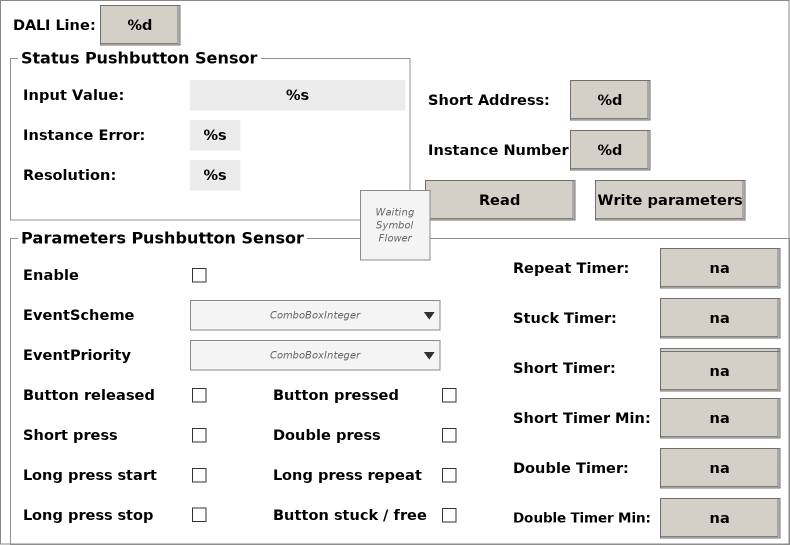
VISUALIZATION Visu_Part301PushButton  // 790x545
    GroupBox (10,230 780x315), "Parameters Pushbutton Sensor"
        Button (650,268 120x40), "%d ms", text variable: DALI_Commissioning.fbPart301PushButton.nDoubleMin
        Button (650,268 120x40), "na", invisible if: Not DALI_Commissioning.fbPart301PushButton.bNoDoubleTimer, input disabled if: Not DALI_Commissioning.fbPart301PushButton.bNoDoubleTimer
        Button (650,168 120x40), "%d ms", text variable: DALI_Commissioning.fbPart301PushButton.nShortMin
        Button (650,168 120x40), "na", invisible if: Not DALI_Commissioning.fbPart301PushButton.bNoRepeatTimer, input disabled if: Not DALI_Commissioning.fbPart301PushButton.bNoRepeatTimer
        Button (650,218 120x40), "%d ms", text variable: DALI_Commissioning.fbPart301PushButton.nDouble
            OnMouseClick: write the text variable via Default, min 0, max 2000, title "Insert value for double timer"
        Button (650,218 120x40), "na", invisible if: Not DALI_Commissioning.fbPart301PushButton.bNoDoubleTimer, input disabled if: Not DALI_Commissioning.fbPart301PushButton.bNoDoubleTimer
        Button (650,118 120x40), "%d ms", text variable: DALI_Commissioning.fbPart301PushButton.nShort
            OnMouseClick: write the text variable via Default, min 10, max 500, title "Insert value for short timer"
        Button (650,121 120x40), "na", invisible if: Not DALI_Commissioning.fbPart301PushButton.bNoRepeatTimer, input disabled if: Not DALI_Commissioning.fbPart301PushButton.bNoRepeatTimer
        Button (650,68 120x40), "%d s", text variable: DALI_Commissioning.fbPart301PushButton.nStuck
            OnMouseClick: write the text variable via Default, min 5, max 255, title "Insert value for stuck timer"
        Button (650,68 120x40), "na", invisible if: Not DALI_Commissioning.fbPart301PushButton.bNoRepeatTimer, input disabled if: Not DALI_Commissioning.fbPart301PushButton.bNoRepeatTimer
        Button (650,18 120x40), "%d ms", text variable: DALI_Commissioning.fbPart301PushButton.nRepeat
            OnMouseClick: write the text variable via Default, min 100, max 2000, title "Insert value for repeat timer"
        Button (650,18 120x40), "na", invisible if: Not DALI_Commissioning.fbPart301PushButton.bNoRepeatTimer, input disabled if: Not DALI_Commissioning.fbPart301PushButton.bNoRepeatTimer
        Textfield (500,23 145x30), "Repeat Timer:"
        Textfield (500,73 145x30), "Stuck Timer:"
        Textfield (500,123 145x30), "Short Timer:"
        Textfield (500,223 145x30), "Double Timer:"
        Textfield (10,30 170x30), "Enable"
        Checkbox (180,30 30x30), variable: DALI_Commissioning.fbPart301PushButton.bEnable
        Textfield (10,70 170x30), "EventScheme"
        Textfield (10,150 170x30), "Button released"
        Textfield (10,190 170x30), "Short press"
        Textfield (10,230 170x30), "Long press start"
        Textfield (10,270 170x30), "Long press stop"
        Textfield (260,150 170x30), "Button pressed"
        Textfield (260,190 170x30), "Double press"
        Textfield (260,230 170x30), "Long press repeat"
        Textfield (260,270 170x30), "Button stuck / free"
        Checkbox (180,150 30x30), variable: DALI_Commissioning.fbPart301PushButton.bButtonReleased
        Checkbox (180,190 30x30), variable: DALI_Commissioning.fbPart301PushButton.bShortPress
        Checkbox (180,230 30x30), variable: DALI_Commissioning.fbPart301PushButton.bLongPressStart
        Checkbox (430,150 30x30), variable: DALI_Commissioning.fbPart301PushButton.bButtonPressed
        Checkbox (430,190 30x30), variable: DALI_Commissioning.fbPart301PushButton.bDoublePress
        Checkbox (430,230 29x30), variable: DALI_Commissioning.fbPart301PushButton.bLongPressRepeat
        Checkbox (430,270 30x30), variable: DALI_Commissioning.fbPart301PushButton.bButtonStuck
        ComboBoxInteger (180,70 250x30), variable: DALI_Commissioning.fbPart301PushButton.eEventScheme, text list: 'EventScheme'
        Checkbox (180,270 28x29), variable: DALI_Commissioning.fbPart301PushButton.bLongPressStop
        Textfield (10,110 170x30), "EventPriority"
        ComboBoxInteger (180,110 250x30), variable: DALI_Commissioning.fbPart301PushButton.eEventPriority, text list: 'EventPriority'
        Textfield (500,173 145x30), "Short Timer Min:"
        Textfield (500,273 145x30), "Double Timer Min:"
    GroupBox (10,50 400x170), "Status Pushbutton Sensor"
        Textfield (10,30 160x30), "Input Value:"
        Textfield (10,70 160x30), "Instance Error:"
        Textfield (10,110 160x30), "Resolution:"
        Textfield (180,30 215x30), "%s", text variable: DALI_Commissioning.fbPart301PushButton.sInputValue
        Textfield (180,70 50x30), "%s", text variable: DALI_Commissioning.fbPart301PushButton.nInstanceError
        Textfield (180,110 50x30), "%s", text variable: DALI_Commissioning.fbPart301PushButton.nResolution
    Button (425,180 150x40), "Read"
        OnMouseClick: execute { DALI_Commissioning.fbPart301PushButton.bRead := TRUE; }
    WaitingSymbolFlower (360,190 70x70), invisible if: DALI_Commissioning.fbPart301PushButton.bHideWaitSymbol
    Button (595,180 150x40), "Write parameters"
        OnMouseClick: execute { DALI_Commissioning.fbPart301PushButton.bWrite := TRUE; }
    Group (10,5 170x40)
        Textfield (0,0 110x40), "DALI Line:"
        Button (90,0 80x40), "%d", text variable: GVL_Internal.nDALILine
            OnMouseClick: write the text variable via Default, min 1, max 10, title "Choose line"
    Textfield (425,80 160x40), "Short Address:"
    Button (570,80 80x40), "%d", text variable: DALI_Commissioning.fbPart301PushButton.nAddress
        OnMouseClick: write the text variable via Default, min 0, max 63, title "Insert Short Address"
    Textfield (425,130 150x40), "Instance Number:"
    Button (570,130 80x40), "%d", text variable: DALI_Commissioning.fbPart301PushButton.nInstanceAddress
        OnMouseClick: write the text variable via Default, min 0, max 31, title "Insert instance number"
END_VISUALIZATION

(* stored: Version 1.1.0.1, ProductVersion 3.1.4024.12
   Visu Visu_Part301PushButton: Id {2b0b9e9a-ce66-464b-855a-c342ef06fc4a} *)
